// Library/POUs/Write/MC_WriteAnalogOutput/Structures/WriteAnalogOutputSendData
{attribute 'pack_mode' := '1'}
// ------------------------------------------------------------------------- 
//  SRCI Robot Library                                                
// ------------------------------------------------------------------------- 
//                                                                           
//  Object:      MoveLinearAbsoluteSendData                                       
//  Author:      Thorsten Brach                                                
//  Date:        2024-07-30
//
//  Description:                                              
//   
//                                                                           
//  Copyright: 
//    (C) 2024 Thorsten Brach. All rights reserved                                                                                                                                            
//             Licensed under the LGPL-3.0 license.
//                                                                           
//  Disclaimer:                                                                           
//    This project is provided without any guarantee and can be used for   
//    private and commercial purposes. Any use is at the user’s 
//    own risk and responsibility.
//
// -------------------------------------------------------------------------
TYPE WriteAnalogOutputSendData EXTENDS CmdHeader: 
STRUCT
  /// ID of Action that will be executed when this command is active
  /// • >0: Start Action - Start executing the Action function with the identical ListenerID.
  /// • <0: Stop Action  -  Stop executing the Action function with the identical ListenerID.
  /// • 0: No trigger (default)-  If no EmitterID is defined, the function will not trigger any Action during its execution
  /// For more information see section Triggers of this chapter or chapter 5.5.12.4.
  EmitterID          : ARRAY [0..3] OF SINT;
  /// Reserve
  Reserve            : BYTE;
  /// ID of associated trigger function:
  /// •  0: No Trigger (default)  No trigger related behavior
  /// • >0: Trigger - Start executing when the trigger function with the identical EmitterID is triggered.
  /// Always positive.
  /// For more information, see chapter 5.5.12 Triggers
  ListenerID         : SINT;
  /// Number of the analog input 1..32
  Index              : USINT;
  /// Unit of set Value:
  Unit               : USINT;
  /// Value of analog output
  Value              : REAL;
END_STRUCT
END_TYPE

// Library/POUs/Write/MC_WriteDigitalOutputs/Structures/WriteDigitalOutputsOutCmd
{attribute 'pack_mode' := '1'} 
// ------------------------------------------------------------------------- 
//  SRCI Robot Library                                                
// ------------------------------------------------------------------------- 
//                                                                           
//  Object:      WriteDigitalOutputsOutCmd                                       
//  Author:      Thorsten Brach                                                
//  Date:        2024-08-08
//
//  Description:                                              
//   
//                                                                           
//  Copyright: 
//    (C) 2024 Thorsten Brach. All rights reserved                                                                                                                                            
//             Licensed under the LGPL-3.0 license.
//                                                                           
//  Disclaimer:                                                                           
//    This project is provided without any guarantee and can be used for   
//    private and commercial purposes. Any use is at the user’s 
//    own risk and responsibility.
//
// -------------------------------------------------------------------------
TYPE WriteDigitalOutputsOutCmd :
STRUCT
  /// Unique system-generated ID of the "Action" when the function is triggered.
  /// • >0: The "Action" is started by the trigger function with identical FollowID.
  /// • <0: The "Action" is stopped by the trigger function with identical FollowID.
  /// For more information see chapter 5.5.12.4.
  OriginID           : INT;
  /// Relates to ListenerID >0 
  /// Number of successful trigger -based command invocations
  /// For more information refer to chapter 5.5.12.4.
  InvocationCounter  : USINT;
END_STRUCT
END_TYPE

// Library/POUs/Write/MC_WriteDigitalOutputs/Structures/WriteDigitalOutputsParCmd
{attribute 'pack_mode' := '1'} 
// ------------------------------------------------------------------------- 
//  SRCI Robot Library                                                
// ------------------------------------------------------------------------- 
//                                                                           
//  Object:      WriteDigitalOutputsParCmd                                       
//  Author:      Thorsten Brach                                                
//  Date:        2024-08-08
//
//  Description:                                              
//   
//                                                                           
//  Copyright: 
//    (C) 2024 Thorsten Brach. All rights reserved                                                                                                                                            
//             Licensed under the LGPL-3.0 license.
//                                                                           
//  Disclaimer:                                                                           
//    This project is provided without any guarantee and can be used for   
//    private and commercial purposes. Any use is at the user’s 
//    own risk and responsibility.
//
// -------------------------------------------------------------------------
TYPE WriteDigitalOutputsParCmd :
STRUCT
  /// Specifies the desired byte addresses that shall be read
  Index              : ARRAY[0..4] OF USINT;
  /// Specifies which outputs may be written
  OutputBitmask      : ARRAY[0..4] OF BYTE;
  /// Array value of Digital Output
  Values             : ARRAY[0..4] OF BYTE;
  /// Set TRUE to prioritize the execution of this command in the defined target sequence.             
  HighPriority       : BOOL;
  /// ID of associated trigger function:
  /// •  0: No Trigger (default)  No trigger related behavior
  /// • >0: Trigger - Start executing when the trigger function with the identical EmitterID is triggered.
  /// Always positive.
  /// For more information, see chapter 5.5.12 Triggers
  ListenerID         : SINT;
END_STRUCT
END_TYPE

// Library/POUs/Write/MC_WriteDigitalOutputs/Structures/WriteDigitalOutputsRecvData
{attribute 'pack_mode' := '1'} 
// ------------------------------------------------------------------------- 
//  SRCI Robot Library                                                
// ------------------------------------------------------------------------- 
//                                                                           
//  Object:      WriteDigitalOutputsRecvData                                       
//  Author:      Thorsten Brach                                                
//  Date:        2024-08-08
//
//  Description:                                              
//   
//                                                                           
//  Copyright: 
//    (C) 2024 Thorsten Brach. All rights reserved                                                                                                                                            
//             Licensed under the LGPL-3.0 license.
//                                                                           
//  Disclaimer:                                                                           
//    This project is provided without any guarantee and can be used for   
//    private and commercial purposes. Any use is at the user’s 
//    own risk and responsibility.
//
// -------------------------------------------------------------------------
TYPE WriteDigitalOutputsRecvData EXTENDS RspHeader :
STRUCT
  /// Relates to ListenerID >0
  /// Number of successful trigger-based command invocations - For more information refer TO chapter 5.5.12.4
  InvocationCounter : USINT;  
  /// Reserve
  Reserve           : SINT;
  /// Unique system-generated ID of the "Action" when the function is triggered.
  /// • >0: The "Action" is started by the trigger funcrion with identical FollowID.
  /// • <0: The "Action" is stopped by the trigger function with identical FollowID.
  /// For more information see chapter 5.5.12.4 EmitterID, ListenerID, FollowID and OriginID
  OriginID          : INT;
END_STRUCT
END_TYPE

// Library/POUs/Write/MC_WriteDigitalOutputs/Structures/WriteDigitalOutputsSendData
{attribute 'pack_mode' := '1'}
// ------------------------------------------------------------------------- 
//  SRCI Robot Library                                                
// ------------------------------------------------------------------------- 
//                                                                           
//  Object:      WriteDigitalOutputsSendData                                       
//  Author:      Thorsten Brach                                                
//  Date:        2024-08-08
//
//  Description:                                              
//   
//                                                                           
//  Copyright: 
//    (C) 2024 Thorsten Brach. All rights reserved                                                                                                                                            
//             Licensed under the LGPL-3.0 license.
//                                                                           
//  Disclaimer:                                                                           
//    This project is provided without any guarantee and can be used for   
//    private and commercial purposes. Any use is at the user’s 
//    own risk and responsibility.
//
// -------------------------------------------------------------------------
TYPE WriteDigitalOutputsSendData EXTENDS CmdHeader: 
STRUCT
  /// ID of Action that will be executed when this command is active
  /// • >0: Start Action - Start executing the Action function with the identical ListenerID.
  /// • <0: Stop Action  -  Stop executing the Action function with the identical ListenerID.
  /// • 0: No trigger (default)-  If no EmitterID is defined, the function will not trigger any Action during its execution
  /// For more information see section Triggers of this chapter or chapter 5.5.12.4.
  EmitterID          : ARRAY [0..3] OF SINT;
  /// ID of associated trigger function:
  /// •  0: No Trigger (default)  No trigger related behavior
  /// • >0: Trigger - Start executing when the trigger function with the identical EmitterID is triggered.
  /// Always positive.
  /// For more information, see chapter 5.5.12 Triggers
  ListenerID         : SINT;
  /// Reserve
  Reserve            : BYTE;
  /// Specifies the desired byte addresses that shall be read
  Index              : ARRAY[0..4] OF USINT;
  /// Specifies which outputs may be written
  OutputBitmask      : ARRAY[0..4] OF BYTE;
  /// Array value of Digital Output
  Values             : ARRAY[0..4] OF BYTE;
END_STRUCT
END_TYPE

// Library/POUs/Write/MC_WriteFrameData/Structures/WriteFrameDataOutCmd
{attribute 'pack_mode' := '1'} 
// ------------------------------------------------------------------------- 
//  SRCI Robot Library                                                
// ------------------------------------------------------------------------- 
//                                                                           
//  Object:      WriteFrameDataOutCmd                                       
//  Author:      Thorsten Brach                                                
//  Date:        2024-08-08
//
//  Description:                                              
//   
//                                                                           
//  Copyright: 
//    (C) 2024 Thorsten Brach. All rights reserved                                                                                                                                            
//             Licensed under the LGPL-3.0 license.
//                                                                           
//  Disclaimer:                                                                           
//    This project is provided without any guarantee and can be used for   
//    private and commercial purposes. Any use is at the user’s 
//    own risk and responsibility.
//
// -------------------------------------------------------------------------
TYPE WriteFrameDataOutCmd :
STRUCT
  /// Unique system-generated ID of the "Action" when the function is triggered.
  /// • >0: The "Action" is started by the trigger function with identical FollowID.
  /// • <0: The "Action" is stopped by the trigger function with identical FollowID.
  /// For more information see chapter 5.5.12.4.
  OriginID           : INT;
  /// Relates to ListenerID >0 
  /// Number of successful trigger -based command invocations
  /// For more information refer to chapter 5.5.12.4.
  InvocationCounter  : USINT;
END_STRUCT
END_TYPE

// Library/POUs/Write/MC_WriteFrameData/Structures/WriteFrameDataParCmd
{attribute 'pack_mode' := '1'} 
// ------------------------------------------------------------------------- 
//  SRCI Robot Library                                                
// ------------------------------------------------------------------------- 
//                                                                           
//  Object:      WriteFrameDataParCmd                                       
//  Author:      Thorsten Brach                                                
//  Date:        2024-08-08
//
//  Description:                                              
//   
//                                                                           
//  Copyright: 
//    (C) 2024 Thorsten Brach. All rights reserved                                                                                                                                            
//             Licensed under the LGPL-3.0 license.
//                                                                           
//  Disclaimer:                                                                           
//    This project is provided without any guarantee and can be used for   
//    private and commercial purposes. Any use is at the user’s 
//    own risk and responsibility.
//
// -------------------------------------------------------------------------
TYPE WriteFrameDataParCmd :
STRUCT
  /// Frame index M
  /// • 0: WCS (default) O
  /// • 1..254: UCS (User frames)
  FrameNo            : USINT;
  /// Frame data (see chapter 5.5.6.2)
  FrameData          : FrameData;
END_STRUCT
END_TYPE

// Library/POUs/Write/MC_WriteFrameData/Structures/WriteFrameDataRecvData
{attribute 'pack_mode' := '1'} 
// ------------------------------------------------------------------------- 
//  SRCI Robot Library                                                
// ------------------------------------------------------------------------- 
//                                                                           
//  Object:      WriteFrameDataRecvData                                       
//  Author:      Thorsten Brach                                                
//  Date:        2024-08-08
//
//  Description:                                              
//   
//                                                                           
//  Copyright: 
//    (C) 2024 Thorsten Brach. All rights reserved                                                                                                                                            
//             Licensed under the LGPL-3.0 license.
//                                                                           
//  Disclaimer:                                                                           
//    This project is provided without any guarantee and can be used for   
//    private and commercial purposes. Any use is at the user’s 
//    own risk and responsibility.
//
// -------------------------------------------------------------------------
TYPE WriteFrameDataRecvData EXTENDS RspHeader :
STRUCT

END_STRUCT
END_TYPE

// Library/POUs/Write/MC_WriteFrameData/Structures/WriteFrameDataSendData
{attribute 'pack_mode' := '1'}
// ------------------------------------------------------------------------- 
//  SRCI Robot Library                                                
// ------------------------------------------------------------------------- 
//                                                                           
//  Object:      WriteFrameDataSendData                                       
//  Author:      Thorsten Brach                                                
//  Date:        2024-08-08
//
//  Description:                                              
//   
//                                                                           
//  Copyright: 
//    (C) 2024 Thorsten Brach. All rights reserved                                                                                                                                            
//             Licensed under the LGPL-3.0 license.
//                                                                           
//  Disclaimer:                                                                           
//    This project is provided without any guarantee and can be used for   
//    private and commercial purposes. Any use is at the user’s 
//    own risk and responsibility.
//
// -------------------------------------------------------------------------
TYPE WriteFrameDataSendData EXTENDS CmdHeader: 
STRUCT
  /// Reserve
  Reserve            : BYTE;
  /// Frame data (see chapter 5.5.6.2)
  FrameData          : FrameData;
  /// Frame index M
  /// • 0: WCS (default) O
  /// • 1..254: UCS (User frames)
  FrameNo            : USINT;
END_STRUCT
END_TYPE

// Library/POUs/Write/MC_WriteIntegers/Structures/WriteIntegersOutCmd
{attribute 'pack_mode' := '1'} 
// ------------------------------------------------------------------------- 
//  SRCI Robot Library                                                
// ------------------------------------------------------------------------- 
//                                                                           
//  Object:      WriteIntegersOutCmd                                       
//  Author:      Thorsten Brach                                                
//  Date:        2024-08-08
//
//  Description:                                              
//   
//                                                                           
//  Copyright: 
//    (C) 2024 Thorsten Brach. All rights reserved                                                                                                                                            
//             Licensed under the LGPL-3.0 license.
//                                                                           
//  Disclaimer:                                                                           
//    This project is provided without any guarantee and can be used for   
//    private and commercial purposes. Any use is at the user’s 
//    own risk and responsibility.
//
// -------------------------------------------------------------------------
TYPE WriteIntegersOutCmd :
STRUCT
  /// Unique system-generated ID of the "Action" when the function is triggered.
  /// • >0: The "Action" is started by the trigger function with identical FollowID.
  /// • <0: The "Action" is stopped by the trigger function with identical FollowID.
  /// For more information see chapter 5.5.12.4.
  OriginID           : INT;
  /// Relates to ListenerID >0 
  /// Number of successful trigger -based command invocations
  /// For more information refer to chapter 5.5.12.4.
  InvocationCounter  : USINT;
END_STRUCT
END_TYPE

// Library/POUs/Write/MC_WriteIntegers/Structures/WriteIntegersParCmd
{attribute 'pack_mode' := '1'} 
// ------------------------------------------------------------------------- 
//  SRCI Robot Library                                                
// ------------------------------------------------------------------------- 
//                                                                           
//  Object:      WriteIntegersParCmd                                       
//  Author:      Thorsten Brach                                                
//  Date:        2024-08-08
//
//  Description:                                              
//   
//                                                                           
//  Copyright: 
//    (C) 2024 Thorsten Brach. All rights reserved                                                                                                                                            
//             Licensed under the LGPL-3.0 license.
//                                                                           
//  Disclaimer:                                                                           
//    This project is provided without any guarantee and can be used for   
//    private and commercial purposes. Any use is at the user’s 
//    own risk and responsibility.
//
// -------------------------------------------------------------------------
TYPE WriteIntegersParCmd :
STRUCT
  /// Specifies the desired target values that shall be written
  Index              : ARRAY[0..6] OF USINT; 
  /// Array value of integers
  Values             : ARRAY[0..6] OF INT;
  /// Set TRUE to prioritize the execution of this command in the defined target sequence.
  HighPriority       : BOOL;
  /// ID of associated trigger function:
  /// •  0: No Trigger (default)  No trigger related behavior
  /// • >0: Trigger - Start executing when the trigger function with the identical EmitterID is triggered.
  /// Always positive.
  /// For more information, see chapter 5.5.12 Triggers
  ListenerID         : SINT;
END_STRUCT
END_TYPE

// Library/POUs/Write/MC_WriteIntegers/Structures/WriteIntegersRecvData
{attribute 'pack_mode' := '1'} 
// ------------------------------------------------------------------------- 
//  SRCI Robot Library                                                
// ------------------------------------------------------------------------- 
//                                                                           
//  Object:      WriteIntegersRecvData                                       
//  Author:      Thorsten Brach                                                
//  Date:        2024-08-08
//
//  Description:                                              
//   
//                                                                           
//  Copyright: 
//    (C) 2024 Thorsten Brach. All rights reserved                                                                                                                                            
//             Licensed under the LGPL-3.0 license.
//                                                                           
//  Disclaimer:                                                                           
//    This project is provided without any guarantee and can be used for   
//    private and commercial purposes. Any use is at the user’s 
//    own risk and responsibility.
//
// -------------------------------------------------------------------------
TYPE WriteIntegersRecvData EXTENDS RspHeader :
STRUCT
  /// Relates to ListenerID >0
  /// Number of successful trigger-based command invocations - For more information refer TO chapter 5.5.12.4
  InvocationCounter : USINT;  
  /// Reserve
  Reserve           : SINT;
  /// Unique system-generated ID of the "Action" when the function is triggered.
  /// • >0: The "Action" is started by the trigger funcrion with identical FollowID.
  /// • <0: The "Action" is stopped by the trigger function with identical FollowID.
  /// For more information see chapter 5.5.12.4 EmitterID, ListenerID, FollowID and OriginID
  OriginID          : INT;
END_STRUCT
END_TYPE

// Library/POUs/Write/MC_WriteIntegers/Structures/WriteIntegersSendData
{attribute 'pack_mode' := '1'}
// ------------------------------------------------------------------------- 
//  SRCI Robot Library                                                
// ------------------------------------------------------------------------- 
//                                                                           
//  Object:      WriteIntegersSendData                                       
//  Author:      Thorsten Brach                                                
//  Date:        2024-08-08
//
//  Description:                                              
//   
//                                                                           
//  Copyright: 
//    (C) 2024 Thorsten Brach. All rights reserved                                                                                                                                            
//             Licensed under the LGPL-3.0 license.
//                                                                           
//  Disclaimer:                                                                           
//    This project is provided without any guarantee and can be used for   
//    private and commercial purposes. Any use is at the user’s 
//    own risk and responsibility.
//
// -------------------------------------------------------------------------
TYPE WriteIntegersSendData EXTENDS CmdHeader: 
STRUCT
  /// ID of Action that will be executed when this command is active
  /// • >0: Start Action - Start executing the Action function with the identical ListenerID.
  /// • <0: Stop Action  -  Stop executing the Action function with the identical ListenerID.
  /// • 0: No trigger (default)-  If no EmitterID is defined, the function will not trigger any Action during its execution
  /// For more information see section Triggers of this chapter or chapter 5.5.12.4.
  EmitterID          : ARRAY [0..3] OF SINT;
  /// ID of associated trigger function:
  /// •  0: No Trigger (default)  No trigger related behavior
  /// • >0: Trigger - Start executing when the trigger function with the identical EmitterID is triggered.
  /// Always positive.
  /// For more information, see chapter 5.5.12 Triggers
  ListenerID         : SINT;
  /// Reserve
  Reserve            : BYTE;
  /// Specifies the desired target values that shall be written
  Index              : ARRAY[0..6] OF USINT; 
  /// Array value of integers
  Values             : ARRAY[0..6] OF INT;
END_STRUCT
END_TYPE

// Library/POUs/Write/MC_WriteLoadData/Structures/WriteLoadDataOutCmd
{attribute 'pack_mode' := '1'} 
// ------------------------------------------------------------------------- 
//  SRCI Robot Library                                                
// ------------------------------------------------------------------------- 
//                                                                           
//  Object:      WriteLoadDataOutCmd                                       
//  Author:      Thorsten Brach                                                
//  Date:        2024-08-08
//
//  Description:                                              
//   
//                                                                           
//  Copyright: 
//    (C) 2024 Thorsten Brach. All rights reserved                                                                                                                                            
//             Licensed under the LGPL-3.0 license.
//                                                                           
//  Disclaimer:                                                                           
//    This project is provided without any guarantee and can be used for   
//    private and commercial purposes. Any use is at the user’s 
//    own risk and responsibility.
//
// -------------------------------------------------------------------------
TYPE WriteLoadDataOutCmd :
STRUCT
  /// Unique system-generated ID of the "Action" when the function is triggered.
  /// • >0: The "Action" is started by the trigger function with identical FollowID.
  /// • <0: The "Action" is stopped by the trigger function with identical FollowID.
  /// For more information see chapter 5.5.12.4.
  OriginID           : INT;
  /// Relates to ListenerID >0 
  /// Number of successful trigger -based command invocations
  /// For more information refer to chapter 5.5.12.4.
  InvocationCounter  : USINT;
END_STRUCT
END_TYPE

// Library/POUs/Write/MC_WriteLoadData/Structures/WriteLoadDataParCmd
{attribute 'pack_mode' := '1'} 
// ------------------------------------------------------------------------- 
//  SRCI Robot Library                                                
// ------------------------------------------------------------------------- 
//                                                                           
//  Object:      WriteLoadDataParCmd                                       
//  Author:      Thorsten Brach                                                
//  Date:        2024-08-08
//
//  Description:                                              
//   
//                                                                           
//  Copyright: 
//    (C) 2024 Thorsten Brach. All rights reserved                                                                                                                                            
//             Licensed under the LGPL-3.0 license.
//                                                                           
//  Disclaimer:                                                                           
//    This project is provided without any guarantee and can be used for   
//    private and commercial purposes. Any use is at the user’s 
//    own risk and responsibility.
//
// -------------------------------------------------------------------------
TYPE WriteLoadDataParCmd :
STRUCT
  /// Specifies the desired target values that shall be written
  /// Load index
  /// •      0: (default) - Not possible to write
  /// • 1..254: Load data
  LoadNo             : USINT;
  /// Load data (see chapter 5.5.6.4)
  LoadData           : LoadData;
END_STRUCT
END_TYPE

// Library/POUs/Write/MC_WriteLoadData/Structures/WriteLoadDataRecvData
{attribute 'pack_mode' := '1'} 
// ------------------------------------------------------------------------- 
//  SRCI Robot Library                                                
// ------------------------------------------------------------------------- 
//                                                                           
//  Object:      WriteLoadDataRecvData                                       
//  Author:      Thorsten Brach                                                
//  Date:        2024-08-08
//
//  Description:                                              
//   
//                                                                           
//  Copyright: 
//    (C) 2024 Thorsten Brach. All rights reserved                                                                                                                                            
//             Licensed under the LGPL-3.0 license.
//                                                                           
//  Disclaimer:                                                                           
//    This project is provided without any guarantee and can be used for   
//    private and commercial purposes. Any use is at the user’s 
//    own risk and responsibility.
//
// -------------------------------------------------------------------------
TYPE WriteLoadDataRecvData EXTENDS RspHeader :
STRUCT

END_STRUCT
END_TYPE

// Library/POUs/Write/MC_WriteLoadData/Structures/WriteLoadDataSendData
{attribute 'pack_mode' := '1'}
// ------------------------------------------------------------------------- 
//  SRCI Robot Library                                                
// ------------------------------------------------------------------------- 
//                                                                           
//  Object:      WriteLoadDataSendData                                       
//  Author:      Thorsten Brach                                                
//  Date:        2024-08-08
//
//  Description:                                              
//   
//                                                                           
//  Copyright: 
//    (C) 2024 Thorsten Brach. All rights reserved                                                                                                                                            
//             Licensed under the LGPL-3.0 license.
//                                                                           
//  Disclaimer:                                                                           
//    This project is provided without any guarantee and can be used for   
//    private and commercial purposes. Any use is at the user’s 
//    own risk and responsibility.
//
// -------------------------------------------------------------------------
TYPE WriteLoadDataSendData EXTENDS CmdHeader: 
STRUCT
  /// Specifies the desired target values that shall be written
  /// Load index
  /// •      0: (default) - Not possible to write
  /// • 1..254: Load data
  LoadNo             : USINT;
  /// Load data (see chapter 5.5.6.4)
  LoadData           : LoadData;
END_STRUCT
END_TYPE

// Library/POUs/Write/MC_WriteReals/Structures/WriteRealsOutCmd
{attribute 'pack_mode' := '1'} 
// ------------------------------------------------------------------------- 
//  SRCI Robot Library                                                
// ------------------------------------------------------------------------- 
//                                                                           
//  Object:      WriteRealsOutCmd                                       
//  Author:      Thorsten Brach                                                
//  Date:        2024-08-08
//
//  Description:                                              
//   
//                                                                           
//  Copyright: 
//    (C) 2024 Thorsten Brach. All rights reserved                                                                                                                                            
//             Licensed under the LGPL-3.0 license.
//                                                                           
//  Disclaimer:                                                                           
//    This project is provided without any guarantee and can be used for   
//    private and commercial purposes. Any use is at the user’s 
//    own risk and responsibility.
//
// -------------------------------------------------------------------------
TYPE WriteRealsOutCmd :
STRUCT
  /// Unique system-generated ID of the "Action" when the function is triggered.
  /// • >0: The "Action" is started by the trigger function with identical FollowID.
  /// • <0: The "Action" is stopped by the trigger function with identical FollowID.
  /// For more information see chapter 5.5.12.4.
  OriginID           : INT;
  /// Relates to ListenerID >0 
  /// Number of successful trigger -based command invocations
  /// For more information refer to chapter 5.5.12.4.
  InvocationCounter  : USINT;
END_STRUCT
END_TYPE

// Library/POUs/Write/MC_WriteReals/Structures/WriteRealsParCmd
{attribute 'pack_mode' := '1'} 
// ------------------------------------------------------------------------- 
//  SRCI Robot Library                                                
// ------------------------------------------------------------------------- 
//                                                                           
//  Object:      WriteRealsParCmd                                       
//  Author:      Thorsten Brach                                                
//  Date:        2024-08-08
//
//  Description:                                              
//   
//                                                                           
//  Copyright: 
//    (C) 2024 Thorsten Brach. All rights reserved                                                                                                                                            
//             Licensed under the LGPL-3.0 license.
//                                                                           
//  Disclaimer:                                                                           
//    This project is provided without any guarantee and can be used for   
//    private and commercial purposes. Any use is at the user’s 
//    own risk and responsibility.
//
// -------------------------------------------------------------------------
TYPE WriteRealsParCmd :
STRUCT
  /// Specifies the desired target values that shall be written
  Index              : ARRAY[0..6] OF USINT; 
  /// Array value of reas
  Values             : ARRAY[0..6] OF REAL;
  /// Set TRUE to prioritize the execution of this command in the defined target sequence.
  HighPriority       : BOOL;
  /// ID of associated trigger function:
  /// •  0: No Trigger (default)  No trigger related behavior
  /// • >0: Trigger - Start executing when the trigger function with the identical EmitterID is triggered.
  /// Always positive.
  /// For more information, see chapter 5.5.12 Triggers
  ListenerID         : SINT;
END_STRUCT
END_TYPE

// Library/POUs/Write/MC_WriteReals/Structures/WriteRealsRecvData
{attribute 'pack_mode' := '1'} 
// ------------------------------------------------------------------------- 
//  SRCI Robot Library                                                
// ------------------------------------------------------------------------- 
//                                                                           
//  Object:      WriteRealsRecvData                                       
//  Author:      Thorsten Brach                                                
//  Date:        2024-08-08
//
//  Description:                                              
//   
//                                                                           
//  Copyright: 
//    (C) 2024 Thorsten Brach. All rights reserved                                                                                                                                            
//             Licensed under the LGPL-3.0 license.
//                                                                           
//  Disclaimer:                                                                           
//    This project is provided without any guarantee and can be used for   
//    private and commercial purposes. Any use is at the user’s 
//    own risk and responsibility.
//
// -------------------------------------------------------------------------
TYPE WriteRealsRecvData EXTENDS RspHeader :
STRUCT
  /// Relates to ListenerID >0
  /// Number of successful trigger-based command invocations - For more information refer TO chapter 5.5.12.4
  InvocationCounter : USINT;  
  /// Reserve
  Reserve           : SINT;
  /// Unique system-generated ID of the "Action" when the function is triggered.
  /// • >0: The "Action" is started by the trigger funcrion with identical FollowID.
  /// • <0: The "Action" is stopped by the trigger function with identical FollowID.
  /// For more information see chapter 5.5.12.4 EmitterID, ListenerID, FollowID and OriginID
  OriginID          : INT;
END_STRUCT
END_TYPE

// Library/POUs/Write/MC_WriteReals/Structures/WriteRealsSendData
{attribute 'pack_mode' := '1'}
// ------------------------------------------------------------------------- 
//  SRCI Robot Library                                                
// ------------------------------------------------------------------------- 
//                                                                           
//  Object:      WriteRealsSendData                                       
//  Author:      Thorsten Brach                                                
//  Date:        2024-08-08
//
//  Description:                                              
//   
//                                                                           
//  Copyright: 
//    (C) 2024 Thorsten Brach. All rights reserved                                                                                                                                            
//             Licensed under the LGPL-3.0 license.
//                                                                           
//  Disclaimer:                                                                           
//    This project is provided without any guarantee and can be used for   
//    private and commercial purposes. Any use is at the user’s 
//    own risk and responsibility.
//
// -------------------------------------------------------------------------
TYPE WriteRealsSendData EXTENDS CmdHeader: 
STRUCT
  /// ID of Action that will be executed when this command is active
  /// • >0: Start Action - Start executing the Action function with the identical ListenerID.
  /// • <0: Stop Action  -  Stop executing the Action function with the identical ListenerID.
  /// • 0: No trigger (default)-  If no EmitterID is defined, the function will not trigger any Action during its execution
  /// For more information see section Triggers of this chapter or chapter 5.5.12.4.
  EmitterID          : ARRAY [0..3] OF SINT;
  /// ID of associated trigger function:
  /// •  0: No Trigger (default)  No trigger related behavior
  /// • >0: Trigger - Start executing when the trigger function with the identical EmitterID is triggered.
  /// Always positive.
  /// For more information, see chapter 5.5.12 Triggers
  ListenerID         : SINT;
  /// Reserve
  Reserve            : BYTE;
  /// Specifies the desired target values that shall be written
  Index              : ARRAY[0..6] OF USINT; 
  /// Array value of reas
  Values             : ARRAY[0..6] OF REAL;
END_STRUCT
END_TYPE

// Library/POUs/Write/MC_WriteRobotDefaultDynamics/Structures/WriteRobotDefaultDynamicsOutCmd
{attribute 'pack_mode' := '1'} 
// ------------------------------------------------------------------------- 
//  SRCI Robot Library                                                
// ------------------------------------------------------------------------- 
//                                                                           
//  Object:      WriteRobotDefaultDynamicsOutCmd                                       
//  Author:      Thorsten Brach                                                
//  Date:        2024-08-08
//
//  Description:                                              
//   
//                                                                           
//  Copyright: 
//    (C) 2024 Thorsten Brach. All rights reserved                                                                                                                                            
//             Licensed under the LGPL-3.0 license.
//                                                                           
//  Disclaimer:                                                                           
//    This project is provided without any guarantee and can be used for   
//    private and commercial purposes. Any use is at the user’s 
//    own risk and responsibility.
//
// -------------------------------------------------------------------------
TYPE WriteRobotDefaultDynamicsOutCmd :
STRUCT
  /// Commanded dynamics values according to Table 6-141.
  DefaultDynamicValues   : DefaultDynamics;
END_STRUCT
END_TYPE

// Library/POUs/Write/MC_WriteRobotDefaultDynamics/Structures/WriteRobotDefaultDynamicsParCmd
{attribute 'pack_mode' := '1'} 
// ------------------------------------------------------------------------- 
//  SRCI Robot Library                                                
// ------------------------------------------------------------------------- 
//                                                                           
//  Object:      WriteRobotDefaultDynamicsParCmd                                       
//  Author:      Thorsten Brach                                                
//  Date:        2024-08-08
//
//  Description:                                              
//   
//                                                                           
//  Copyright: 
//    (C) 2024 Thorsten Brach. All rights reserved                                                                                                                                            
//             Licensed under the LGPL-3.0 license.
//                                                                           
//  Disclaimer:                                                                           
//    This project is provided without any guarantee and can be used for   
//    private and commercial purposes. Any use is at the user’s 
//    own risk and responsibility.
//
// -------------------------------------------------------------------------
TYPE WriteRobotDefaultDynamicsParCmd :
STRUCT
  /// Default dynamics values according to Table 6-141.
  DynamicValues          : DefaultDynamics;
END_STRUCT
END_TYPE

// Library/POUs/Write/MC_WriteRobotDefaultDynamics/Structures/WriteRobotDefaultDynamicsRecvData
{attribute 'pack_mode' := '1'} 
// ------------------------------------------------------------------------- 
//  SRCI Robot Library                                                
// ------------------------------------------------------------------------- 
//                                                                           
//  Object:      WriteRobotDefaultDynamicsRecvData                                       
//  Author:      Thorsten Brach                                                
//  Date:        2024-08-08
//
//  Description:                                              
//   
//                                                                           
//  Copyright: 
//    (C) 2024 Thorsten Brach. All rights reserved                                                                                                                                            
//             Licensed under the LGPL-3.0 license.
//                                                                           
//  Disclaimer:                                                                           
//    This project is provided without any guarantee and can be used for   
//    private and commercial purposes. Any use is at the user’s 
//    own risk and responsibility.
//
// -------------------------------------------------------------------------
TYPE WriteRobotDefaultDynamicsRecvData EXTENDS RspHeader :
STRUCT
  /// Maximum velocity for the axes.
  /// Range [%]: 
  /// •  <0% : Use default velocity given by the user
  /// •   0% : Use internal minimal velocity
  /// • 100% : Use the entire reference velocity, given by the user
  VelocityRate     : UINT;
  /// Maximum acceleration.
  /// Range [%]:
  /// •  <0% : Use default acceleration given by the user
  /// •   0% : Use internal minimal acceleration
  /// • 100% : Use the entire reference acceleration, given by the user
  AccelerationRate : UINT;
  /// Maximum deceleration.
  /// Range [%] : 
  /// •  <0% : Use default deceleration given by the user
  /// •   0% : Use internal minimal deceleration
  /// • 100% : Use the entire reference deceleration, given by the user
  DecelerationRate : UINT;
  /// Maximum jerk
  /// Range [%] : 
  /// •  <0% : Use default jerk given by the user
  /// •   0% : Use internal minimal jerk
  /// • 100% : Use the entire reference jerk, given by the user (Trapezoidal if possible) 
  JerkRate         : UINT;  
END_STRUCT
END_TYPE

// Library/POUs/Write/MC_WriteRobotDefaultDynamics/Structures/WriteRobotDefaultDynamicsSendData
{attribute 'pack_mode' := '1'}
// ------------------------------------------------------------------------- 
//  SRCI Robot Library                                                
// ------------------------------------------------------------------------- 
//                                                                           
//  Object:      WriteRobotDefaultDynamicsSendData                                       
//  Author:      Thorsten Brach                                                
//  Date:        2024-08-08
//
//  Description:                                              
//   
//                                                                           
//  Copyright: 
//    (C) 2024 Thorsten Brach. All rights reserved                                                                                                                                            
//             Licensed under the LGPL-3.0 license.
//                                                                           
//  Disclaimer:                                                                           
//    This project is provided without any guarantee and can be used for   
//    private and commercial purposes. Any use is at the user’s 
//    own risk and responsibility.
//
// -------------------------------------------------------------------------
TYPE WriteRobotDefaultDynamicsSendData EXTENDS CmdHeader: 
STRUCT
  /// Timestamp
  Timestamp        : IEC_TIMESTAMP;
  /// Maximum velocity for the axes.
  /// Range [%]: 
  /// •  <0% : Use default velocity given by the user
  /// •   0% : Use internal minimal velocity
  /// • 100% : Use the entire reference velocity, given by the user
  VelocityRate     : UINT;
  /// Maximum acceleration.
  /// Range [%]:
  /// •  <0% : Use default acceleration given by the user
  /// •   0% : Use internal minimal acceleration
  /// • 100% : Use the entire reference acceleration, given by the user
  AccelerationRate : UINT;
  /// Maximum deceleration.
  /// Range [%] : 
  /// •  <0% : Use default deceleration given by the user
  /// •   0% : Use internal minimal deceleration
  /// • 100% : Use the entire reference deceleration, given by the user
  DecelerationRate : UINT;
  /// Maximum jerk
  /// Range [%] : 
  /// •  <0% : Use default jerk given by the user
  /// •   0% : Use internal minimal jerk
  /// • 100% : Use the entire reference jerk, given by the user (Trapezoidal if possible) 
  JerkRate         : UINT;  
END_STRUCT
END_TYPE

// Library/POUs/Write/MC_WriteRobotReferenceDynamics/Structures/WriteRobotReferenceDynamicsOutCmd
{attribute 'pack_mode' := '1'} 
// ------------------------------------------------------------------------- 
//  SRCI Robot Library                                                
// ------------------------------------------------------------------------- 
//                                                                           
//  Object:      WriteRobotReferenceDynamicsOutCmd                                       
//  Author:      Thorsten Brach                                                
//  Date:        2024-08-08
//
//  Description:                                              
//   
//                                                                           
//  Copyright: 
//    (C) 2024 Thorsten Brach. All rights reserved                                                                                                                                            
//             Licensed under the LGPL-3.0 license.
//                                                                           
//  Disclaimer:                                                                           
//    This project is provided without any guarantee and can be used for   
//    private and commercial purposes. Any use is at the user’s 
//    own risk and responsibility.
//
// -------------------------------------------------------------------------
TYPE WriteRobotReferenceDynamicsOutCmd :
STRUCT
  /// Commanded reference dynamics values according to Table 6-134
  ReferenceDynamicValues : ReferenceDynamics;
END_STRUCT
END_TYPE

// Library/POUs/Write/MC_WriteRobotReferenceDynamics/Structures/WriteRobotReferenceDynamicsParCmd
{attribute 'pack_mode' := '1'} 
// ------------------------------------------------------------------------- 
//  SRCI Robot Library                                                
// ------------------------------------------------------------------------- 
//                                                                           
//  Object:      WriteRobotReferenceDynamicsParCmd                                       
//  Author:      Thorsten Brach                                                
//  Date:        2024-08-08
//
//  Description:                                              
//   
//                                                                           
//  Copyright: 
//    (C) 2024 Thorsten Brach. All rights reserved                                                                                                                                            
//             Licensed under the LGPL-3.0 license.
//                                                                           
//  Disclaimer:                                                                           
//    This project is provided without any guarantee and can be used for   
//    private and commercial purposes. Any use is at the user’s 
//    own risk and responsibility.
//
// -------------------------------------------------------------------------
TYPE WriteRobotReferenceDynamicsParCmd :
STRUCT
  /// Reference dynamics values according TO Table 6-134.
  DynamicValues : ReferenceDynamics;
END_STRUCT
END_TYPE

// Library/POUs/Write/MC_WriteRobotReferenceDynamics/Structures/WriteRobotReferenceDynamicsRecvData
{attribute 'pack_mode' := '1'} 
// ------------------------------------------------------------------------- 
//  SRCI Robot Library                                                
// ------------------------------------------------------------------------- 
//                                                                           
//  Object:      WriteRobotReferenceDynamicsRecvData                                       
//  Author:      Thorsten Brach                                                
//  Date:        2024-08-08
//
//  Description:                                              
//   
//                                                                           
//  Copyright: 
//    (C) 2024 Thorsten Brach. All rights reserved                                                                                                                                            
//             Licensed under the LGPL-3.0 license.
//                                                                           
//  Disclaimer:                                                                           
//    This project is provided without any guarantee and can be used for   
//    private and commercial purposes. Any use is at the user’s 
//    own risk and responsibility.
//
// -------------------------------------------------------------------------
TYPE WriteRobotReferenceDynamicsRecvData EXTENDS RspHeader :
STRUCT
  /// Commanded reference dynamics values according to Table 6-134
  ReferenceDynamicValues : ReferenceDynamics;
END_STRUCT
END_TYPE

// Library/POUs/Write/MC_WriteRobotReferenceDynamics/Structures/WriteRobotReferenceDynamicsSendData
{attribute 'pack_mode' := '1'}
// ------------------------------------------------------------------------- 
//  SRCI Robot Library                                                
// ------------------------------------------------------------------------- 
//                                                                           
//  Object:      WriteRobotReferenceDynamicsSendData                                       
//  Author:      Thorsten Brach                                                
//  Date:        2024-08-08
//
//  Description:                                              
//   
//                                                                           
//  Copyright: 
//    (C) 2024 Thorsten Brach. All rights reserved                                                                                                                                            
//             Licensed under the LGPL-3.0 license.
//                                                                           
//  Disclaimer:                                                                           
//    This project is provided without any guarantee and can be used for   
//    private and commercial purposes. Any use is at the user’s 
//    own risk and responsibility.
//
// -------------------------------------------------------------------------
TYPE WriteRobotReferenceDynamicsSendData EXTENDS CmdHeader: 
STRUCT
  
  DynamicValues : ReferenceDynamics;
(*
  /// Timestamp
  Timestamp             : IEC_TIMESTAMP;
  /// Path velocity [mm/s](tangent) at 100%
  /// • <0: (default) - Do not change values
  /// • ≥0: Change values according to input value
  VelocityReference     : UINT;
  /// Path acceleration [mm/s2] at 100%
  /// • <0: (default) - Do not change values
  /// • ≥0: Change values according to input value
  AccelerationReference : UINT;
  /// Path deceleration [mm/s2] at 100%
  /// • <0: (default) - Do not change values
  /// • ≥0: Change values according to input value
  DecelerationReference : UINT;
  /// Jerk [mm/s3] at 100%
  /// • <0: (default) - Do not change values
  /// • ≥0: Change values according to input value
  JerkReference        : UINT;
*)
END_STRUCT
END_TYPE

// Library/POUs/Write/MC_WriteRobotSWLimits/Structures/WriteRobotSWLimitsOutCmd
{attribute 'pack_mode' := '1'} 
// ------------------------------------------------------------------------- 
//  SRCI Robot Library                                                
// ------------------------------------------------------------------------- 
//                                                                           
//  Object:      WriteRobotSWLimitsOutCmd                                       
//  Author:      Thorsten Brach                                                
//  Date:        2024-08-08
//
//  Description:                                              
//   
//                                                                           
//  Copyright: 
//    (C) 2024 Thorsten Brach. All rights reserved                                                                                                                                            
//             Licensed under the LGPL-3.0 license.
//                                                                           
//  Disclaimer:                                                                           
//    This project is provided without any guarantee and can be used for   
//    private and commercial purposes. Any use is at the user’s 
//    own risk and responsibility.
//
// -------------------------------------------------------------------------
TYPE WriteRobotSWLimitsOutCmd :
STRUCT
  /// TRUE, when Software limits were overwritten but not activated on RC until a restart of the RC
  RestartRequested       : BOOL;
END_STRUCT
END_TYPE

// Library/POUs/Write/MC_WriteRobotSWLimits/Structures/WriteRobotSWLimitsParCmd
{attribute 'pack_mode' := '1'} 
// ------------------------------------------------------------------------- 
//  SRCI Robot Library                                                
// ------------------------------------------------------------------------- 
//                                                                           
//  Object:      WriteRobotSWLimitsParCmd                                       
//  Author:      Thorsten Brach                                                
//  Date:        2024-08-08
//
//  Description:                                              
//   
//                                                                           
//  Copyright: 
//    (C) 2024 Thorsten Brach. All rights reserved                                                                                                                                            
//             Licensed under the LGPL-3.0 license.
//                                                                           
//  Disclaimer:                                                                           
//    This project is provided without any guarantee and can be used for   
//    private and commercial purposes. Any use is at the user’s 
//    own risk and responsibility.
//
// -------------------------------------------------------------------------
TYPE WriteRobotSWLimitsParCmd :
STRUCT
  /// Limits for joints and external axes according to Table 6-180.
  LimitValues            : SWLimits;
  /// Reset limits to RC specific factory settings
  ResetToFactoryDefaults : BOOL;;
END_STRUCT
END_TYPE

// Library/POUs/Write/MC_WriteRobotSWLimits/Structures/WriteRobotSWLimitsRecvData
{attribute 'pack_mode' := '1'} 
// ------------------------------------------------------------------------- 
//  SRCI Robot Library                                                
// ------------------------------------------------------------------------- 
//                                                                           
//  Object:      WriteRobotSWLimitsRecvData                                       
//  Author:      Thorsten Brach                                                
//  Date:        2024-08-08
//
//  Description:                                              
//   
//                                                                           
//  Copyright: 
//    (C) 2024 Thorsten Brach. All rights reserved                                                                                                                                            
//             Licensed under the LGPL-3.0 license.
//                                                                           
//  Disclaimer:                                                                           
//    This project is provided without any guarantee and can be used for   
//    private and commercial purposes. Any use is at the user’s 
//    own risk and responsibility.
//
// -------------------------------------------------------------------------
TYPE WriteRobotSWLimitsRecvData EXTENDS RspHeader :
STRUCT
  /// TRUE, when Software limits were overwritten but not activated on RC until a restart of the RC
  RestartRequested       : BOOL;
END_STRUCT
END_TYPE

// Library/POUs/Write/MC_WriteRobotSWLimits/Structures/WriteRobotSWLimitsSendData
{attribute 'pack_mode' := '1'}
// ------------------------------------------------------------------------- 
//  SRCI Robot Library                                                
// ------------------------------------------------------------------------- 
//                                                                           
//  Object:      WriteRobotSWLimitsSendData                                       
//  Author:      Thorsten Brach                                                
//  Date:        2024-08-08
//
//  Description:                                              
//   
//                                                                           
//  Copyright: 
//    (C) 2024 Thorsten Brach. All rights reserved                                                                                                                                            
//             Licensed under the LGPL-3.0 license.
//                                                                           
//  Disclaimer:                                                                           
//    This project is provided without any guarantee and can be used for   
//    private and commercial purposes. Any use is at the user’s 
//    own risk and responsibility.
//
// -------------------------------------------------------------------------
TYPE WriteRobotSWLimitsSendData EXTENDS CmdHeader: 
STRUCT
  /// Limits for joints and external axes according to Table 6-180.
  LimitValues            : SWLimits;
  /// Reset limits to RC specific factory settings
  ResetToFactoryDefaults : BOOL;;
END_STRUCT
END_TYPE

// Library/POUs/Write/MC_WriteSystemVariable/Structures/WriteSystemVariableOutCmd
{attribute 'pack_mode' := '1'} 
// ------------------------------------------------------------------------- 
//  SRCI Robot Library                                                
// ------------------------------------------------------------------------- 
//                                                                           
//  Object:      WriteSystemVariableOutCmd                                       
//  Author:      Thorsten Brach                                                
//  Date:        2024-08-08
//
//  Description:                                              
//   
//                                                                           
//  Copyright: 
//    (C) 2024 Thorsten Brach. All rights reserved                                                                                                                                            
//             Licensed under the LGPL-3.0 license.
//                                                                           
//  Disclaimer:                                                                           
//    This project is provided without any guarantee and can be used for   
//    private and commercial purposes. Any use is at the user’s 
//    own risk and responsibility.
//
// -------------------------------------------------------------------------
TYPE WriteSystemVariableOutCmd :
STRUCT
  /// Unique system-generated ID of the "Action" when the function is triggered.
  /// • >0: The "Action" is started by the trigger function with identical FollowID.
  /// • <0: The "Action" is stopped by the trigger function with identical FollowID.
  /// For more information see chapter 5.5.12.4 EmitterID, ListenerID, FollowID and OriginID
  OriginID           : INT;
  /// Relates to ListenerID >0
  /// Number of successful trigger -based command invocations
  /// For more information refer to chapter 5.5.12.4.
  InvocationCounter  : USINT;
  /// TRUE, when Software limits were overwritten but not activated on RC until a restart of the RC
  RestartRequested       : BOOL;
END_STRUCT
END_TYPE

// Library/POUs/Write/MC_WriteSystemVariable/Structures/WriteSystemVariableParCmd
{attribute 'pack_mode' := '1'} 
// ------------------------------------------------------------------------- 
//  SRCI Robot Library                                                
// ------------------------------------------------------------------------- 
//                                                                           
//  Object:      WriteSystemVariableParCmd                                       
//  Author:      Thorsten Brach                                                
//  Date:        2024-08-08
//
//  Description:                                              
//   
//                                                                           
//  Copyright: 
//    (C) 2024 Thorsten Brach. All rights reserved                                                                                                                                            
//             Licensed under the LGPL-3.0 license.
//                                                                           
//  Disclaimer:                                                                           
//    This project is provided without any guarantee and can be used for   
//    private and commercial purposes. Any use is at the user’s 
//    own risk and responsibility.
//
// -------------------------------------------------------------------------
TYPE WriteSystemVariableParCmd :
STRUCT
  /// Defines the parameter list which should be used:
  /// • FALSE: Standardized parameter list (default):
  ///          -  Read parameters on the RC based on a standardized parameter list
  /// • TRUE: Manufacturer specific parameter list:
  ///        -  Read parameters on the RC based on robot manufacturers-specific parameter lists
  RCParameter        : BOOL;
  /// Requested parameter ID in selected parameter list.
  /// •          0: undefined (default)
  /// • 1..65 535: Parameter ID
  ParameterID        : ARRAY[0..7] OF UINT;
  /// ID of the requested sub parameter in selected parameter list.
  /// • 0: ID 0 (default) (relates only to parameters without sub parameters)
  /// • 1..255: Indices 1 to 255 (relates only to parameters with sub parameters)
  SubParameterID     : ARRAY[0..7] OF USINT;  
  /// Parameter data type as specified in Table 6-621.
  DataType           : ARRAY[0..7] OF USINT;
  /// Parameter data addressed by input values of ParameterID[0] and SubParameterID[0]
  Data_0             : ARRAY[0..3] OF BYTE;
  /// Parameter data addressed by input values of ParameterID[1] and SubParameterID[1]
  Data_1             : ARRAY[0..3] OF BYTE;
  /// Parameter data addressed by input values of ParameterID[2] and SubParameterID[2]
  Data_2             : ARRAY[0..3] OF BYTE;
  /// Parameter data addressed by input values of ParameterID[3] and SubParameterID[3]
  Data_3             : ARRAY[0..3] OF BYTE;
  /// Parameter data addressed by input values of ParameterID[4] and SubParameterID[4]
  Data_4             : ARRAY[0..3] OF BYTE;
  /// Parameter data addressed by input values of ParameterID[5] and SubParameterID[5]
  Data_5             : ARRAY[0..3] OF BYTE;
  /// Parameter data addressed by input values of ParameterID[6] and SubParameterID[6]
  Data_6             : ARRAY[0..3] OF BYTE;
  /// Parameter data addressed by input values of ParameterID[7] and SubParameterID[7]
  Data_7             : ARRAY[0..3] OF BYTE;
  /// ID of associated trigger function:
  /// •  0: No Trigger (default)  No trigger related behavior
  /// • >0: Trigger - Start executing when the trigger function with the identical EmitterID is triggered.
  /// Always positive.
  /// For more information, see chapter 5.5.12 Triggers
  ListenerID         : SINT;
END_STRUCT
END_TYPE

// Library/POUs/Write/MC_WriteSystemVariable/Structures/WriteSystemVariableRecvData
{attribute 'pack_mode' := '1'} 
// ------------------------------------------------------------------------- 
//  SRCI Robot Library                                                
// ------------------------------------------------------------------------- 
//                                                                           
//  Object:      WriteSystemVariableRecvData                                       
//  Author:      Thorsten Brach                                                
//  Date:        2024-08-08
//
//  Description:                                              
//   
//                                                                           
//  Copyright: 
//    (C) 2024 Thorsten Brach. All rights reserved                                                                                                                                            
//             Licensed under the LGPL-3.0 license.
//                                                                           
//  Disclaimer:                                                                           
//    This project is provided without any guarantee and can be used for   
//    private and commercial purposes. Any use is at the user’s 
//    own risk and responsibility.
//
// -------------------------------------------------------------------------
TYPE WriteSystemVariableRecvData EXTENDS RspHeader :
STRUCT
  /// Relates to ListenerID >0
  /// Number of successful trigger-based command invocations - For more information refer TO chapter 5.5.12.4
  InvocationCounter : USINT;  
  /// Reserve
  Reserve           : SINT;
  /// Unique system-generated ID of the "Action" when the function is triggered.
  /// • >0: The "Action" is started by the trigger funcrion with identical FollowID.
  /// • <0: The "Action" is stopped by the trigger function with identical FollowID.
  /// For more information see chapter 5.5.12.4 EmitterID, ListenerID, FollowID and OriginID
  OriginID          : INT;
  /// TRUE, when Software limits were overwritten but not activated on RC until a restart of the RC
  RestartRequested  : BOOL;
END_STRUCT
END_TYPE

// Library/POUs/Write/MC_WriteSystemVariable/Structures/WriteSystemVariableSendData
{attribute 'pack_mode' := '1'}
// ------------------------------------------------------------------------- 
//  SRCI Robot Library                                                
// ------------------------------------------------------------------------- 
//                                                                           
//  Object:      WriteSystemVariableSendData                                       
//  Author:      Thorsten Brach                                                
//  Date:        2024-08-08
//
//  Description:                                              
//   
//                                                                           
//  Copyright: 
//    (C) 2024 Thorsten Brach. All rights reserved                                                                                                                                            
//             Licensed under the LGPL-3.0 license.
//                                                                           
//  Disclaimer:                                                                           
//    This project is provided without any guarantee and can be used for   
//    private and commercial purposes. Any use is at the user’s 
//    own risk and responsibility.
//
// -------------------------------------------------------------------------
TYPE WriteSystemVariableSendData EXTENDS CmdHeader: 
STRUCT
  /// ID of Action that will be executed when this command is active
  /// • >0: Start Action - Start executing the Action function with the identical ListenerID.
  /// • <0: Stop Action  -  Stop executing the Action function with the identical ListenerID.
  /// • 0: No trigger (default)-  If no EmitterID is defined, the function will not trigger any Action during its execution
  /// For more information see section Triggers of this chapter or chapter 5.5.12.4.
  EmitterID          : ARRAY [0..3] OF SINT;
  /// ID of associated trigger function:
  /// •  0: No Trigger (default)  No trigger related behavior
  /// • >0: Trigger - Start executing when the trigger function with the identical EmitterID is triggered.
  /// Always positive.
  /// For more information, see chapter 5.5.12 Triggers
  ListenerID         : SINT;  
  /// Reserve
  Reserve            : BYTE;
  /// Requested parameter ID in selected parameter list.
  /// •          0: undefined (default)
  /// • 1..65 535: Parameter ID
  ParameterID        : ARRAY[0..7] OF UINT;
  /// ID of the requested sub parameter in selected parameter list.
  /// • 0: ID 0 (default) (relates only to parameters without sub parameters)
  /// • 1..255: Indices 1 to 255 (relates only to parameters with sub parameters)
  SubParameterID     : ARRAY[0..7] OF USINT;  
  /// Parameter data type as specified in Table 6-621.
  DataType           : ARRAY[0..7] OF USINT;
  /// Parameter data addressed by input values of ParameterID[0] and SubParameterID[0]
  Data_0             : ARRAY[0..3] OF BYTE;
  /// Parameter data addressed by input values of ParameterID[1] and SubParameterID[1]
  Data_1             : ARRAY[0..3] OF BYTE;
  /// Parameter data addressed by input values of ParameterID[2] and SubParameterID[2]
  Data_2             : ARRAY[0..3] OF BYTE;
  /// Parameter data addressed by input values of ParameterID[3] and SubParameterID[3]
  Data_3             : ARRAY[0..3] OF BYTE;
  /// Parameter data addressed by input values of ParameterID[4] and SubParameterID[4]
  Data_4             : ARRAY[0..3] OF BYTE;
  /// Parameter data addressed by input values of ParameterID[5] and SubParameterID[5]
  Data_5             : ARRAY[0..3] OF BYTE;
  /// Parameter data addressed by input values of ParameterID[6] and SubParameterID[6]
  Data_6             : ARRAY[0..3] OF BYTE;
  /// Parameter data addressed by input values of ParameterID[7] and SubParameterID[7]
  Data_7             : ARRAY[0..3] OF BYTE;
  /// • FALSE: Standardized parameter list (default):
  ///          -  Read parameters on the RC based on a standardized parameter list
  /// • TRUE: Manufacturer specific parameter list:
  ///        -  Read parameters on the RC based on robot manufacturers-specific parameter lists
  RCParameter        : BOOL;
END_STRUCT
END_TYPE

// Library/POUs/Write/MC_WriteToolData/Structures/WriteToolDataOutCmd
{attribute 'pack_mode' := '1'} 
// ------------------------------------------------------------------------- 
//  SRCI Robot Library                                                
// ------------------------------------------------------------------------- 
//                                                                           
//  Object:      WriteToolDataOutCmd                                       
//  Author:      Thorsten Brach                                                
//  Date:        2024-08-08
//
//  Description:                                              
//   
//                                                                           
//  Copyright: 
//    (C) 2024 Thorsten Brach. All rights reserved                                                                                                                                            
//             Licensed under the LGPL-3.0 license.
//                                                                           
//  Disclaimer:                                                                           
//    This project is provided without any guarantee and can be used for   
//    private and commercial purposes. Any use is at the user’s 
//    own risk and responsibility.
//
// -------------------------------------------------------------------------
TYPE WriteToolDataOutCmd :
STRUCT
END_STRUCT
END_TYPE

// Library/POUs/Write/MC_WriteToolData/Structures/WriteToolDataParCmd
{attribute 'pack_mode' := '1'} 
// ------------------------------------------------------------------------- 
//  SRCI Robot Library                                                
// ------------------------------------------------------------------------- 
//                                                                           
//  Object:      WriteToolDataParCmd                                       
//  Author:      Thorsten Brach                                                
//  Date:        2024-08-08
//
//  Description:                                              
//   
//                                                                           
//  Copyright: 
//    (C) 2024 Thorsten Brach. All rights reserved                                                                                                                                            
//             Licensed under the LGPL-3.0 license.
//                                                                           
//  Disclaimer:                                                                           
//    This project is provided without any guarantee and can be used for   
//    private and commercial purposes. Any use is at the user’s 
//    own risk and responsibility.
//
// -------------------------------------------------------------------------
TYPE WriteToolDataParCmd :
STRUCT
  /// Tool index
  /// •      0: Flange (default) Not possible to change
  /// • 1..254: Tool Frame
  ToolNo            : USINT;
  /// Tool data (see chapter 5.5.6.3)
  ToolData          : ToolData;
END_STRUCT
END_TYPE

// Library/POUs/Write/MC_WriteToolData/Structures/WriteToolDataRecvData
{attribute 'pack_mode' := '1'} 
// ------------------------------------------------------------------------- 
//  SRCI Robot Library                                                
// ------------------------------------------------------------------------- 
//                                                                           
//  Object:      WriteToolDataRecvData                                       
//  Author:      Thorsten Brach                                                
//  Date:        2024-08-08
//
//  Description:                                              
//   
//                                                                           
//  Copyright: 
//    (C) 2024 Thorsten Brach. All rights reserved                                                                                                                                            
//             Licensed under the LGPL-3.0 license.
//                                                                           
//  Disclaimer:                                                                           
//    This project is provided without any guarantee and can be used for   
//    private and commercial purposes. Any use is at the user’s 
//    own risk and responsibility.
//
// -------------------------------------------------------------------------
TYPE WriteToolDataRecvData EXTENDS RspHeader :
STRUCT
END_STRUCT
END_TYPE

// Library/POUs/Write/MC_WriteToolData/Structures/WriteToolDataSendData
{attribute 'pack_mode' := '1'}
// ------------------------------------------------------------------------- 
//  SRCI Robot Library                                                
// ------------------------------------------------------------------------- 
//                                                                           
//  Object:      WriteToolDataSendData                                       
//  Author:      Thorsten Brach                                                
//  Date:        2024-08-08
//
//  Description:                                              
//   
//                                                                           
//  Copyright: 
//    (C) 2024 Thorsten Brach. All rights reserved                                                                                                                                            
//             Licensed under the LGPL-3.0 license.
//                                                                           
//  Disclaimer:                                                                           
//    This project is provided without any guarantee and can be used for   
//    private and commercial purposes. Any use is at the user’s 
//    own risk and responsibility.
//
// -------------------------------------------------------------------------
TYPE WriteToolDataSendData EXTENDS CmdHeader: 
STRUCT
  /// Reserve
  Reserve           : BYTE;
  /// Tool index
  /// •      0: Flange (default) Not possible to change
  /// • 1..254: Tool Frame
  ToolNo            : USINT;
  /// Tool data (see chapter 5.5.6.3)
  ToolData          : ToolData;
END_STRUCT
END_TYPE

// Library/Structures/_internal/SplineDataSend
{attribute 'pack_mode' := '1'} 
// ------------------------------------------------------------------------- 
//  SRCI Robot Library                                                
// ------------------------------------------------------------------------- 
//                                                                           
//  Object:      SplineDataSend                                       
//  Author:      Thorsten Brach                                                
//  Date:        2024-08-01
//
//  Description:                                              
//   
//                                                                           
//  Copyright: 
//    (C) 2024 Thorsten Brach. All rights reserved                                                                                                                                            
//             Licensed under the LGPL-3.0 license.
//                                                                           
//  Disclaimer:                                                                           
//    This project is provided without any guarantee and can be used for   
//    private and commercial purposes. Any use is at the user’s 
//    own risk and responsibility.
//
// -------------------------------------------------------------------------
TYPE SplineDataSend :
STRUCT
    /// Absolute target coordinates in the selected coordinate system (see ToolNo and FrameNo).
    Position         : RobotCartesianPosition;
    /// TCP velocity in % of nominal velocity.
    /// •  <0% : Use default velocity (default)
    /// •   0% : Use internal minimal velocity
    /// • 100% : Use maximal reference velocity
    /// • See chapter 5.5.7 Robot dynamics
    VelocityRate     : UINT;    
    /// Acceleration for movement in % of nominal acceleration.
    /// •  <0% : Use default acceleration (default)
    /// •   0% : Use internal minimal acceleration
    /// • 100% : Use maximal reference acceleration
    /// • See chapter 5.5.7 Robot dynamics
    AccelerationRate : UINT;    
    /// Deceleration for movement in % of nominal deceleration.
    /// •  <0% : Use default deceleration (default)
    /// •   0% : Use internal minimal deceleration
    /// • 100% : Use maximal reference deceleration
    /// • See chapter 5.5.7 Robot dynamics
    DecelerationRate : UINT;    
    /// Jerk of the movement in % of nominal jerk.
    /// <0% o Use default jerk (default)
    /// 0% o Use internal minimal jerk
    /// 100% o Use maximal reference jerk
    /// See chapter 5.5.7 Robot dynamics
    JerkRate         : UINT;
    /// Index of tool
    /// 0: Flange (default)
    /// 1..254: Tool frames
    ToolNo           : USINT;    
    /// Index of frame
    /// 0: WCS (default)
    /// 1..254: User frames
    FrameNo          : USINT;    
    /// [ms] Parameter is used if it is greater than 0 (default):
    /// Parameter defines the time for the movement to reach the target position
    /// Velocity input can be ignored
    /// Acceleration, Deceleration and jerk will be ignored
    /// Define two consecutive points with identical positions and specified Time to realize waiting time on spline.
    /// Error is sent by the RC, if the time cannot be kept.
    MoveTime         : UINT;  
END_STRUCT
END_TYPE

// Library/Structures/AxesGroup/Acyclic/AxesGroupAcyclic
{attribute 'pack_mode' := '1'} 
// ------------------------------------------------------------------------- 
//  SRCI Robot Library                                                
// ------------------------------------------------------------------------- 
//                                                                           
//  Object:      AxesGroupAcyclic                                       
//  Author:      Thorsten Brach                                                
//  Date:        2024-06-01
//
//  Description:                                              
//   
//                                                                           
//  Copyright: 
//    (C) 2024 Thorsten Brach. All rights reserved                                                                                                                                            
//             Licensed under the LGPL-3.0 license.
//                                                                           
//  Disclaimer:                                                                           
//    This project is provided without any guarantee and can be used for   
//    private and commercial purposes. Any use is at the user’s 
//    own risk and responsibility.
//
// -------------------------------------------------------------------------
TYPE AxesGroupAcyclic :
STRUCT
  // Active command register 
  ActiveCommandRegister : ActiveCommandRegisterFB;
END_STRUCT
END_TYPE

// Library/Structures/AxesGroup/Acyclic/AxesGroupAcyclicAcrEntry
{attribute 'pack_mode' := '1'} 
// ------------------------------------------------------------------------- 
//  SRCI Robot Library                                                
// ------------------------------------------------------------------------- 
//                                                                           
//  Object:      AxesGroupAcyclicAcrEntry                                       
//  Author:      Thorsten Brach                                                
//  Date:        2024-06-01
//
//  Description:                                              
//   
//                                                                           
//  Copyright: 
//    (C) 2024 Thorsten Brach. All rights reserved                                                                                                                                            
//             Licensed under the LGPL-3.0 license.
//                                                                           
//  Disclaimer:                                                                           
//    This project is provided without any guarantee and can be used for   
//    private and commercial purposes. Any use is at the user’s 
//    own risk and responsibility.
//
// -------------------------------------------------------------------------
TYPE AxesGroupAcyclicAcrEntry :
STRUCT
  /// Unique indentifier 
  UniqueID   : UINT; 
  /// State of the command entry
  State      : ActiveCommandRegisterState;  
  /// Command data ( 1 = DataToSend 2 = DataInBuffer )
  Command    : ARRAY[1..2] OF AxesGroupAcyclicAcrEntryCmdBuffer;
  /// response data ( 1 = DataRecv 2 = DataInRecvBuffer )
  Response   : ARRAY[1..2] OF AxesGroupAcyclicAcrEntryRspBuffer;
  /// Pointer to the corresponding command-FB to enable a callback mechanism
  pCommandFB : POINTER TO RobotLibraryBaseFB;
END_STRUCT
END_TYPE

// Library/Structures/AxesGroup/Acyclic/AxesGroupAcyclicAcrEntryCmd
{attribute 'pack_mode' := '1'} 
// ------------------------------------------------------------------------- 
//  SRCI Robot Library                                                
// ------------------------------------------------------------------------- 
//                                                                           
//  Object:      AxesGroupAcyclicAcrEntryCmd                                       
//  Author:      Thorsten Brach                                                
//  Date:        2024-06-01
//
//  Description:                                              
//   
//                                                                           
//  Copyright: 
//    (C) 2024 Thorsten Brach. All rights reserved                                                                                                                                            
//             Licensed under the LGPL-3.0 license.
//                                                                           
//  Disclaimer:                                                                           
//    This project is provided without any guarantee and can be used for   
//    private and commercial purposes. Any use is at the user’s 
//    own risk and responsibility.
//
// -------------------------------------------------------------------------
TYPE AxesGroupAcyclicAcrEntryCmd :
STRUCT 
  /// Byte 00-03: Command header
  // Header  : AxesGroupAcyclicAcrEntryCmdHeader;
  /// Payload buffer
  Payload    : AxesGroupAcyclicAcrEntryCmdBuffer;  
  /// send buffer
  SendBuffer : AxesGroupAcyclicAcrEntryCmdBuffer;
END_STRUCT
END_TYPE

// Library/Structures/AxesGroup/Acyclic/AxesGroupAcyclicAcrEntryCmdBuffer
{attribute 'pack_mode' := '1'} 
// ------------------------------------------------------------------------- 
//  SRCI Robot Library                                                
// ------------------------------------------------------------------------- 
//                                                                           
//  Object:      AxesGroupAcyclicAcrEntryCmdBuffer                                       
//  Author:      Thorsten Brach                                                
//  Date:        2024-06-01
//
//  Description:                                              
//   
//                                                                           
//  Copyright: 
//    (C) 2024 Thorsten Brach. All rights reserved                                                                                                                                            
//             Licensed under the LGPL-3.0 license.
//                                                                           
//  Disclaimer:                                                                           
//    This project is provided without any guarantee and can be used for   
//    private and commercial purposes. Any use is at the user’s 
//    own risk and responsibility.
//
// -------------------------------------------------------------------------
TYPE AxesGroupAcyclicAcrEntryCmdBuffer :
STRUCT
  /// Timestamp
  Timestamp         : SystemTime;
  /// Buffer state
  State             : BufferStateCmd;
  /// Payload defined by type per CMD definition. Processed by Appl. Layer Task.
  Payload           : ARRAY[0..RobotLibraryParameter.TELEGRAM_PAYLOAD_MAX] OF BYTE;
  /// Payload length
  PayloadLen        : UDINT;  
  /// Payload poiner position   
  PayLoadPtr        : UINT;
END_STRUCT
END_TYPE

// Library/Structures/AxesGroup/Acyclic/AxesGroupAcyclicAcrEntryCmdHeader
{attribute 'pack_mode' := '1'} 
// ------------------------------------------------------------------------- 
//  SRCI Robot Library                                                
// ------------------------------------------------------------------------- 
//                                                                           
//  Object:      AxesGroupAcyclicAcrEntryCmdHeader                                       
//  Author:      Thorsten Brach                                                
//  Date:        2024-06-01
//
//  Description:                                              
//   
//                                                                           
//  Copyright: 
//    (C) 2024 Thorsten Brach. All rights reserved                                                                                                                                            
//             Licensed under the LGPL-3.0 license.
//                                                                           
//  Disclaimer:                                                                           
//    This project is provided without any guarantee and can be used for   
//    private and commercial purposes. Any use is at the user’s 
//    own risk and responsibility.
//
// -------------------------------------------------------------------------
TYPE AxesGroupAcyclicAcrEntryCmdHeader :
STRUCT
  /// Byte 00-01 :  CMD type as per specification
  CmdType      : CmdType;
  /// Byte 02  : ExecutionMode (Bit 0..3)
  ExecMode     : ExecutionMode;  
  /// Byte 03 : CMD priority (Bit 0..3)
  Prio         : PriorityLevel;
  /// Byte 03 : Parameter Sequence (Bit 4..7 )
  ParSeq       : BYTE;
END_STRUCT
END_TYPE

// Library/Structures/AxesGroup/Acyclic/AxesGroupAcyclicAcrEntryCmdTrigger
{attribute 'pack_mode' := '1'} 
// ------------------------------------------------------------------------- 
//  SRCI Robot Library                                                
// ------------------------------------------------------------------------- 
//                                                                           
//  Object:      AxesGroupAcyclicAcrEntryCmdTrigger                                       
//  Author:      Thorsten Brach                                                
//  Date:        2024-06-01
//
//  Description:                                              
//   
//                                                                           
//  Copyright: 
//    (C) 2024 Thorsten Brach. All rights reserved                                                                                                                                            
//             Licensed under the LGPL-3.0 license.
//                                                                           
//  Disclaimer:                                                                           
//    This project is provided without any guarantee and can be used for   
//    private and commercial purposes. Any use is at the user’s 
//    own risk and responsibility.
//
// -------------------------------------------------------------------------
TYPE AxesGroupAcyclicAcrEntryCmdTrigger :
STRUCT
  /// Trigger related EmitterID
  EmitterID    : ARRAY[0..3] OF SINT;
  /// Trigger related ListenerID 
  ListenerID   : SINT;
  /// Reserver
  Reserve      : BYTE;
END_STRUCT
END_TYPE

